// TwinCAT 3 PLC project AD_DA_V2
// ProgramVersion: 3.1.4020.2
// libraries:
//   Tc2_ControllerToolbox, * (Beckhoff Automation GmbH)
//   Tc2_Standard, * (Beckhoff Automation GmbH)
//   Tc2_System, * (Beckhoff Automation GmbH)
//   Tc3_Module, * (Beckhoff Automation GmbH)
//   VisuDialogs, * (System)
// project tree:
//   FB_Lib/Conversion/ FB_ConfigAnalog.TcPOU, FB_Ia.TcPOU, FB_Qa.TcPOU, ST_MinMax.TcDUT
//   FB_Lib/FB_ActionneurSimple/ FB_ActionneurSimple.TcPOU, ST_Erreur.TcDUT, ST_ParamActionneur.TcDUT
//   FB_Lib/ FB_analo_and_digital.TcPOU, FB_Etape.TcPOU
//   FB_Lib/FB_GestionModes/ FB_Btn.TcPOU, FB_CycleAuto.TcPOU, FB_CycleInit.TcPOU, FB_CycleMan.TcPOU, FB_MMA.TcPOU, p_InitVar.TcPOU
//   FB_Lib/FB_GestionModes/IO/ ST_IO.TcDUT, ST_IOInput.TcDUT, ST_IOInputSimul.TcDUT, ST_IOOutput.TcDUT, ST_IOOutputSimul.TcDUT
//   FB_Lib/FB_GestionModes/Param/ E_ModeMMA.TcDUT, ST_Param.TcDUT, ST_ParamFixed.TcDUT, ST_ParamRecipe.TcDUT, ST_ParamStatus.TcDUT
//   / GlobalTextList.TcGTLO, PlcTask.TcTTO, Visualisierungsmanager.TcVMO (not stored)
//   GVLs/ GVL.TcGVL
//   POUs/ MAIN.TcPOU
//   VISUs/ vi_ConvertAnalog.TcVIS, vi_ConvertAnalog_1.TcVIS
// (motion and I/O tree: see PLC project 1calcul)
// real-time tasks:
//   TASK PlcTask: cycle T#1ms, priority 20, ADS port 350
// variable links:
//   AD-DA_V2/AD-DA_V2 Instance <-> Device 2 (EtherCAT)/Box 1 (BK1150)
//     PlcTask Inputs/GVL.fbIa.IaEntree <-> Term 4 (KL3404)/Channel 2/Daten Ein
//     PlcTask Outputs/GVL.fbQa.QaSortie <-> Term 5 (KL4434)/Channel 2/Daten Aus

CONFIGURATION AD_DA_V2
    RESOURCE PLC ON TwinCAT3
        TASK PlcTask(INTERVAL := T#10ms, PRIORITY := 20);
        PROGRAM MAIN WITH PlcTask : MAIN;
    END_RESOURCE
END_CONFIGURATION

// ---- FB_Lib/Conversion/ST_MinMax.TcDUT
TYPE ST_MinMax :
STRUCT
	lrMin: LREAL;
	lrMax: LREAL;
END_STRUCT
END_TYPE

// ---- FB_Lib/FB_ActionneurSimple/ST_Erreur.TcDUT
TYPE ST_Erreur :
STRUCT
	xState:BOOL; 		//shows the current error state
	iId : INT; 			//error number currently active
	sMessage : STRING; 	//error message for the active error
END_STRUCT
END_TYPE

// ---- FB_Lib/FB_ActionneurSimple/ST_ParamActionneur.TcDUT
TYPE ST_ParamActionneur :
STRUCT
	tTimeOut : TIME; 			//max time allowed for moving to position bevor xState=TRUE
	xPresenceSensOut : BOOL; 	//If at the out-pos a Sensor is available
	xPresenceSensIn : BOOL; 	//If at the in-pos a Sensor is availaible
	tMoveOutTimeDelay : TIME; 	//delay after activating xPresenceSensOut before turning off output. When there is no Sensor, only this time will be used.
	tMoveInTimeDelay : TIME; 	//delay after activating xPresenceSensIn before turning off output. When there is no Sensor, only this time will be used.
END_STRUCT
END_TYPE

// ---- FB_Lib/FB_GestionModes/IO/ST_IO.TcDUT
TYPE ST_IO :
STRUCT
	stIn:ST_IOInput;
	stOut:ST_IOOutput;
END_STRUCT
END_TYPE

// ---- FB_Lib/FB_GestionModes/IO/ST_IOInput.TcDUT
TYPE ST_IOInput :
STRUCT
	IxAruIO AT%I*  :BOOL;
	xStartIO AT%I* :BOOL;
	xStopIO AT%I*  :BOOL;
	xResetIO AT%I* :BOOL;
	xAuto AT%I* : BOOL;
	xManual AT%I* : BOOL;
END_STRUCT
END_TYPE

// ---- FB_Lib/FB_GestionModes/IO/ST_IOInputSimul.TcDUT
TYPE ST_IOInputSimul :
STRUCT
	IxAru :BOOL;
END_STRUCT
END_TYPE

// ---- FB_Lib/FB_GestionModes/IO/ST_IOOutput.TcDUT
TYPE ST_IOOutput :
STRUCT
	QxLampeRouge AT%Q*:BOOL;
	QxLampeVerte AT%Q* : BOOL;
	QxLampeOrange AT%Q* :BOOL;
END_STRUCT
END_TYPE

// ---- FB_Lib/FB_GestionModes/IO/ST_IOOutputSimul.TcDUT
TYPE ST_IOOutputSimul :
STRUCT
	QxLampeRouge AT%Q*:BOOL;
END_STRUCT
END_TYPE

// ---- FB_Lib/FB_GestionModes/Param/E_ModeMMA.TcDUT

TYPE E_ModeMMA :
(
	Init := 0,
	Auto,
	Man
);
END_TYPE

// ---- FB_Lib/FB_GestionModes/Param/ST_Param.TcDUT
TYPE ST_Param :
STRUCT
	stStatus:ST_ParamStatus;//informations d'états (compteur de pièces, modes,...)
	stFixed:ST_ParamFixed;//Paramètres pas en lien avec le produit, fixe
	stRecipe:ST_ParamRecipe;//Paramètres en lien avec le produit
END_STRUCT
END_TYPE

// ---- FB_Lib/FB_GestionModes/Param/ST_ParamFixed.TcDUT
TYPE ST_ParamFixed :
STRUCT
END_STRUCT
END_TYPE

// ---- FB_Lib/FB_GestionModes/Param/ST_ParamRecipe.TcDUT
TYPE ST_ParamRecipe :
STRUCT
	
END_STRUCT
END_TYPE

// ---- FB_Lib/FB_GestionModes/Param/ST_ParamStatus.TcDUT
TYPE ST_ParamStatus :
STRUCT
	eMMA : E_ModeMMA; 
	xModePasAPas:BOOL;
	xErreur:BOOL;
	xInitOk:BOOL;//indique que l'initialisation a été exécutée
END_STRUCT
END_TYPE

// ---- GVLs/GVL.TcGVL

VAR_GLOBAL
		fbQa:FB_Qa;
		fbIa:FB_Ia;
END_VAR

// ---- POUs/MAIN.TcPOU
PROGRAM MAIN
VAR
	Consigne: LREAL;
	deltaConsigne :LREAL;
	PID : FB_CTRL_PID;
	
END_VAR

fbQa();
fbIa();




PID.fSetpointValue:=Consigne;
PID.fActualValue:=fbIa.lrValeur;
PID.eMode:=2;

PID(fOut=>fbQa.lrConsigne,stParams.fKp:=2,stParams.tTn:=T#10S,stParams.tTv:=T#10S,stParams.tTd:=T#10S,stParams.fOutMaxLimit:=10,stParams.fOutMinLimit:=-10,stParams.bARWOnIPartOnly:=FALSE,
stParams.bDInTheFeedbackPath:=TRUE,stParams.bPInTheFeedbackPath:=TRUE,stParams.tCtrlCycleTime:=T#10MS,stParams.tTaskCycleTime:=T#10MS);

END_PROGRAM

// ---- FB_Lib/Conversion/FB_Qa.TcPOU
FUNCTION_BLOCK FB_Qa
VAR_INPUT
	///consigne dans l'unité de l'utilisateur, selon min et max de fbCongig.stValeur
	lrConsigne: LREAL;
	///configuration de la sortie analogique
	fbConfig: FB_ConfigAnalog;
END_VAR
VAR_OUTPUT
	///sortie analogique, atention, supprimer MatchingSize lors de la liaison avec la borne
	QaSortie AT %Q*: DINT;
	///écart de précision sur la valeur de consigne => valeur +/- écart
	lrEcart: LREAL;
	///tension en volt
	lrTension: LREAL;
END_VAR

// 
QaSortie:=fbConfig.mConvertValToAn(lrConsigne,lrTension=>lrTension,lrEcart=>lrEcart);

END_FUNCTION_BLOCK

// ---- FB_Lib/Conversion/FB_ConfigAnalog.TcPOU
FUNCTION_BLOCK FB_ConfigAnalog
VAR_INPUT
	///nombre de bit de la variable de transit du bus de terrain
	uiNbreBitBus: UINT;
	///nombre de bit du convertiseur Analogique/digital 
	uiNbreBitConv: UINT;
	///valeur min et max de la tension
	stTension: ST_minMax;
	///valeur min et max de la consigne
	stValeur: ST_minMax;
END_VAR
VAR
	udiNbreIncBus: UDINT;
	lrTemp: LREAL;
	///nombre d'incrément avant décalage d'offset sur valeur de consigne
	lrValInc: LREAL;
END_VAR

METHOD mCalculDelta : LREAL
VAR_INPUT
	stMinMax: ST_MinMax;
END_VAR
mCalculDelta:=stMinMax.lrMax-stMinMax.lrMin;
END_METHOD

METHOD mCalculInc : UDINT
VAR_INPUT
	uiNbreBitBus: UDINT;
END_VAR

mCalculInc:=SHL(1,uiNbreBitBus);
//mCaclulInc:=EXPT(2,uiNbreBitBus);
END_METHOD

METHOD mConvertAnToVal : LREAL
VAR_INPUT
	///valeur de consigne
	lrAna: LREAL;
END_VAR
VAR_OUTPUT
	///tension de la borne de sortie
	lrTension: LREAL;
	///Ecart de l'escalier sur la borne de sortie en unité de valeur
	lrEcart: LREAL;
END_VAR
VAR
	lrValeur: LREAL;
END_VAR
//vérification que lrVal compris entre min et max
(*IF lrVal>stValeur.lrMax THEN
	lrVal:=stValeur.lrMax;
END_IF
IF lrVal>stValeur.lrMin THEN
	lrVal:=stValeur.lrMin;
END_IF*)
(*
lrVal:=MAX(lrVal,stValeur.lrMax);
lrVal:=MIN(lrVal,stValeur.lrMin);
*)


//Calcul du nombre d'incréments
udiNbreIncBus:=mCalculInc(uiNbreBitBus);
//Conversion de la valeur vers le résultat
//deltaTension/Nbreinc <-> deltaVal/Nbreinc val
lrValeur:=0;//réponse = 0 si hors condition
IF mCalculDelta(stValeur)<>0 THEN
	//décalage selon min max de la tension
	//IF stTension.lrMin<0 THEN
	//	//ajout de l'offset si min négatif
	//	lrTemp:=lrValInc-udiNbreIncBus/2-1;
	//	ELSE
	//	lrTemp:=lrValInc;
	//END_IF
	//nombre d'incréments par rapport à lrVal, avec décalage de stValeur.lrMin
	//lrValeur:=(lrAna*mCalculDelta(stValeur)-stValeur.lrMin)/udiNbreIncBus;
	//lrValInc:=udiNbreIncBus*(lrVal-stValeur.lrMin)/mCalculDelta(stValeur);
	//temp:=(iValMax-iValMin) / temp2;
	//oPhysicalValue:=iValMin + (temp * (iRAWValue+temp2/2));
	lrValeur:=(mCalculDelta(stValeur)/udiNbreIncBus)*lrAna;
	
END_IF
//résultat de la méthode
mConvertAnToVal:=lrValeur;
//calcul de l'incrément tension
lrEcart:=(mCalculDelta(stTension)/udiNbreIncBus);
//résultat en unitée de tension
lrTension:=lrValInc*lrEcart+stTension.lrMin;
END_METHOD

METHOD mConvertValToAn : DINT
VAR_INPUT
	///valeur de consigne
	lrVal: LREAL;
END_VAR
VAR_OUTPUT
	///tension de la borne de sortie
	lrTension: LREAL;
	///Ecart de l'escalier sur la borne de sortie en unité de valeur
	lrEcart: LREAL;
END_VAR
//vérification que lrVal compris entre min et max
(*IF lrVal>stValeur.lrMax THEN
	lrVal:=stValeur.lrMax;
END_IF
IF lrVal>stValeur.lrMin THEN
	lrVal:=stValeur.lrMin;
END_IF*)
(*
lrVal:=MAX(lrVal,stValeur.lrMax);
lrVal:=MIN(lrVal,stValeur.lrMin);
*)
lrVal:=LIMIT(stValeur.lrMin,lrVal,stValeur.lrMax);

//Calcul du nombre d'incréments
udiNbreIncBus:=mCalculInc(uiNbreBitBus);
//Conversion de la valeur vers le résultat
//deltaTension/Nbreinc <-> deltaVal/Nbreinc val
lrTemp:=0;//réponse = 0 si hors condition
IF mCalculDelta(stValeur)<>0 THEN
	//nombre d'incréments par rapport à lrVal, avec décalage de stValeur.lrMin
	lrValInc:=udiNbreIncBus*(lrVal-stValeur.lrMin)/mCalculDelta(stValeur);
	//décalage selon min max de la tension
	IF stTension.lrMin<0 THEN
		//ajout de l'offset si min négatif
		lrTemp:=lrValInc-udiNbreIncBus/2-1;
		ELSE
		lrTemp:=lrValInc;
	END_IF
END_IF
//résultat de la méthode
mConvertValToAn:=LREAL_TO_DINT(lrTemp);
//calcul de l'incrément tension
lrEcart:=(mCalculDelta(stTension)/udiNbreIncBus);
//résultat en unitée de tension
lrTension:=lrValInc*lrEcart+stTension.lrMin;
END_METHOD

END_FUNCTION_BLOCK

// ---- FB_Lib/Conversion/FB_Ia.TcPOU
FUNCTION_BLOCK FB_Ia
VAR_INPUT
	///configuration de la sortie analogique
	fbConfig: FB_ConfigAnalog;
END_VAR
VAR_OUTPUT
	///Valeur dans l'unité de l'utilisateur, selon min et max de fbCongig.stValeur
	lrValeur: LREAL;
	///sortie analogique, atention, supprimer MatchingSize lors de la liaison avec la borne
	IaEntree AT%I*: INT;
	///écart de précision sur la valeur de consigne => valeur +/- écart
	lrEcart: LREAL;
	///tension en volt
	lrTension: LREAL;
END_VAR
VAR
END_VAR

lrValeur:=fbConfig.mConvertAnToVal(IaEntree,lrTension=>lrTension,lrEcart=>lrEcart);

END_FUNCTION_BLOCK

// ---- FB_Lib/FB_ActionneurSimple/FB_ActionneurSimple.TcPOU
FUNCTION_BLOCK FB_ActionneurSimple
VAR_INPUT
	xInGoOut AT%I*:BOOL;				//input for going out
	xInGoIn AT%I*:BOOL;					//input for going in
	xReset AT%I*:BOOL;					//Reset all (go back to init state
	
	xAutorizeOut AT%I* : BOOL;		//allowed to do the move requested with xInGoOut, If this is false Programm will threw an error
	xAutorizeIn At%I* : BOOL;			//allowed to do the move requested with xInGoIn, If this is false Programm will threw an error
	
	stParam:ST_ParamActionneur;	//Param for actuator 
END_VAR
VAR_OUTPUT
	xInOutPos:BOOL;
	xInInPos:BOOL;
	
	xGoingOutNow AT%Q*:BOOL; //indication that actor is going in Out-Pos
	xGoingInNow AT%Q*:BOOL; //indication that actor is going in In-Pos
	
	QxOutOutput AT%Q*:BOOL;//Output to actuator for going Out
	QxInOutput AT%Q*:BOOL;//Output to actuator for going In
	
	IxSensOut AT%I*:BOOL;	//Sensor for the reached In-Pos
	IxSensIn AT%I*:BOOL;//Sensor for the reached Out-Pos
		
	stError:ST_Erreur;//Error Struct
	
	QxVanneDeBloquage AT%Q* : BOOL; //Vanne de blocace. Elle devient seulement 1 si l'autorisation entree/sortie est present
END_VAR
VAR
	fbEtape:FB_Etape;
	fbTimeOut:TON;
	fbRTrigOut:R_Trig;
	fbRTrigIn:R_Trig;
		
	

END_VAR

fbEtape.mActualisation(xModeStepForStep,xNextStep);

//check rising edges on 
fbRTrigOut(clk:=xInGoOut);
fbRTrigIn(clk:=xInGoIn);

//Go to the next step when there is an Out-Command
IF fbRTrigOut.Q AND NOT(fbEtape.iNo>=200 AND fbEtape.iNo<=299) THEN	//When rising-edge was detected
	IF xAutorizeOut THEN
		fbEtape.piVal:=200;
	ELSE
		stError.iId:=10;
		stError.sMessage:='Autorisation refusee pour action sortir verin';
	END_IF		
fbEtape.piVal:=200;	
END_IF

//Go to the next step when there is an In-Command
IF fbRTrigIn.Q AND NOT(fbEtape.iNo>=100 AND fbEtape.iNo<=199) THEN	//When rising-edge was detected and not already going In
	IF xAutorizeIn THEN
		fbEtape.piVal:=100;
	ELSE
		stError.iId:=11;
		stError.sMessage:='Autorisation refusee pour action rentrer verin';
	END_IF	
END_IF

//Reset
IF xReset THEN
	fbEtape.piVal:=0;
	stError.xState:=0;
	xInOutPos:=0;
	xInInPos:=0;
END_IF

//check pour vanne de blocage
QxVanneDeBloquage:= (xAutorizeOut OR xAutorizeIn);

//Reset de l'erreur
IF stError.xState THEN
	stError.iId:=0;
	stError.sMessage:='';
END_IF



CASE fbEtape.iNo OF
	0:fbEtape.psMess:='Wait for an In or Out command';
	//-----------------------------------------------
	100:fbEtape.psMess:='Action go In';
		IF xAutorizeIn THEN
			fbEtape.piVal:=110;
			fbEtape.tTimeQ:=stParam.tMoveInTimeDelay;
		END_IF
	110:fbEtape.psMess:='Going in, waiting for IxSensIn';
		IF (IxSensIn AND stParam.xPresenceSensIn) OR NOT stParam.xPresenceSensIn THEN
			fbEtape.piVal:=150;
		END_IF
	150:fbEtape.psMess:='Action rentre, attend tenps d enveloppe';
		IF fbEtape.xTimeQ THEN
			fbEtape.piSVal:=199;
		END_IF
	199:fbEtape.psMess:='In-Position reached';
		IF (NOT IxSensIn) AND stParam.xPresenceSensIn THEN
			fbEtape.piVal:=150;
		END_IF
	//-----------------------------------------------
	200:fbEtape.psMess:='Action go Out';
		IF xAutorizeOut THEN
			fbEtape.piVal:=210;
			fbEtape.tTimeQ:=stParam.tMoveInTimeDelay;
		END_IF
	210:fbEtape.psMess:='Going Out, waiting for IxSensOut';
		IF (IxSensOut AND stParam.xPresenceSensOut) OR NOT stParam.xPresenceSensOut THEN
			fbEtape.piVal:=250;
		END_IF
	250:fbEtape.psMess:='Action sort, attend temps d enveloppe';
		IF fbEtape.xTimeQ THEN
			fbEtape.piSVal:=299;
		END_IF
	299:fbEtape.psMess:='Out-Pos reached';
		IF (NOT IxSensOut) AND stParam.xPresenceSensoUT THEN
			fbEtape.piVal:=250;
		END_IF
	
	999:fbEtape.psMess:='Erreur';
END_CASE

//Activation du Timer
fbTimeOut(IN:=(fbEtape.iNo>100 AND fbEtape.iNo<199 OR fbEtape.iNo>200 AND fbEtape.iNo<299)
				AND (NOT fbRTrigIn.Q AND NOT fbRTrigOut.Q),PT:=stParam.tTimeOut);	


(*Liste des erreurs possibles :
-	10 Si un ordre de déplacement sort est donné et que l’entrée, xAutoriseSort n’est pas vrai, on indique une erreur
-	11 Idem pour xAutoriseRentre
-	20 Erreur de timeout sort
-	21 Erreur de timeout rentre
-	30 Les deux fins de course sont vraies en même temps
-	31 Double consignes, xSetSort=1 et xSetRentre=1*)				
//Gestion des erreurs
IF fbTimeOut.Q THEN
	IF fbEtape.iNo < 200 THEN
		stError.sMessage:='Erreur de timeout rentre';
		stError.iId:=21;
	ELSIF fbEtape.iNo>200 THEN
		stError.sMessage:='Erreur de timeout sort';
		stError.iId:=20;
	END_IF
ELSIF IxSensIn AND IxSensOut THEN
	stError.sMessage:='Les deus fins de course sont vraies en même temps';
	stError.iId:=30;
ELSIF xInGoOut AND xInGoIn THEN
	stError.sMessage:='Double consigne,xSetSort=1 et xSetRentre=1';
	stError.iId:=31;
END_IF

stError.xState :=fbEtape.iNo=999 OR fbTimeOut.Q OR (IxSensIn AND IxSensOut) OR (xInGoIn AND xInGoOut);


//Activation des états
xInInPos:=fbEtape.iNo=199;
xInOutPos:=fbEtape.iNo=299;
xGoingInNow:= QxInOutput AND NOT IxSensIn;
xGoingOutNow:= QxOutOutput AND NOT IxSensOut;


//Activation des sorties
QxOutOutput:=fbEtape.iNo>200 AND fbEtape.iNo<=299;
QxInOutput:=fbEtape.iNo>100 AND fbEtape.iNo<=199;

END_FUNCTION_BLOCK

// ---- FB_Lib/FB_Etape.TcPOU
FUNCTION_BLOCK FB_Etape
VAR_INPUT
	tTimeQ :TIME;			//Time to stay in one state after which xTimeQ will go to TRUE
END_VAR
VAR_OUTPUT
	tTimeState: TIME ; 	//passed time in the actual state
	xTimeQ : BOOL ;		//is TRUE when time passed in the actual State is greather then tTimeQ
	xTransition:BOOL; 	//information that the state has just changed. For use when entering a new State the first time
	iNo:INT:=0; 		//State number running at the moment
	sMess :STRING ; 	//Information message about the current running state
END_VAR
VAR
	iMemNo:INT;				//Used for xTransition. Saves the actual state of the machine
	fbTon:ton;				//Timer for the actual State
	fbRtrig:R_trig;			//detector for rising edges
	xMemModeStepByStep:BOOL;	//Mem for the actual running Mode (see method mActualisation)
	
END_VAR

//executed at each state-machine-loop
METHOD PUBLIC mActualisation
VAR_INPUT
	xModeStepByStep: BOOL; //activate the Stepping-Mode (TRUE=ON)
	xSetNextStep: BOOL; //go to the next Step on rising eddge
END_VAR
//manage StepByStep
//-----------------

//Detect rising edge
fbRtrig(CLK:=xSetNextStep);
//copy the mode input to use it in piSVal
xMemModeStepByStep:=xModeStepByStep;

//detect a state changement in the state machine
xTransition:=iNo<>iMemNo;

//start Method when the state has changed
IF xTransition THEN
	mTransition();
END_IF

//manage the Timer and associated Variabels
//-----------------------------------------
fbTON(IN:=(iNo=iMemNo), PT:=T#71582M47S295MS, ET=>tTimeState); //will be resetted when the state is changed

//going to TRUE when longer in the actual State than tTimeQ
xTimeQ:=(tTimeState>=tTimeQ);

//save the last running state
iMemNo:=iNo;
END_METHOD

//Executed when a State has changed
METHOD PRIVATE mTransition
//make a new String to display
sMess:=CONCAT('iNo:=',int_to_string(iNo));
END_METHOD

//going to the next step while paying attention to StepByStep Mode
PROPERTY PUBLIC piSVal : INT
SET
IF NOT xMemModeStepByStep THEN
	//Step by step mode is off
	iNo:=piSVal;
	ELSIF fbRtrig.Q THEN
		//a button press on "xSetNextStep" has been detected
		iNo:=piSVal;
END_IF
END_SET
END_PROPERTY

//going to the next step without paying attention to StepByStep Mode
PROPERTY PUBLIC piVal : INT
SET
//set the next step
iNo:=piVal;
END_SET
END_PROPERTY

//
PROPERTY PUBLIC psMess : STRING
SET
//write the description of the actual step to sMess
IF xTransition THEN
	sMess:=psMess;
END_IF
END_SET
END_PROPERTY

END_FUNCTION_BLOCK

// ---- FB_Lib/FB_analo_and_digital.TcPOU
FUNCTION_BLOCK FB_analo_and_digital
VAR_INPUT
	iRAWValue : LREAL;			//raw Value read from sensor (registre)
	iResolution : INT; 		//resolution in bits
	iValMin: INT;			//min physical value possible
	iValMax: INT;			//max physical value possible
	iTransToPhysical : BOOL;	//RAW --> Physical when TRUE
	iPhysical2Value: LREAL; 	//valeur physique (ex tr/min)
	iValInputMax: INT;		//max input value at the Box
	iValInputMin: INT;		//min input value at the Box
	iPhysicalValue : LREAL;	//valeur physique sur l'entree de l'input
END_VAR
VAR_OUTPUT
	oValInputMin: INT;		//min input value at the Box
	oPhysicalValue : LREAL;	//valeur physique sur l'entree de l'input
	oInputValue : LREAL;	//valeur physique sur l'entree de l'input
	oPhysical2Value: LREAL; 	//valeur physique (ex tr/min)
	oRAWValue : LREAL;			//raw Value read from sensor (registre)
END_VAR
VAR	
	temp : LREAL;
	temp2 : LREAL;	
END_VAR

temp2:=expt(2,iResolution);



IF(iTransToPhysical) THEN
	//RAW Input to physical value
	temp:=(iValInputMax-iValInputMin) / temp2;
	oInputValue:=iValInputMin + (temp * (iRAWValue + temp2/2));
	
	
	temp:=(iValMax-iValMin) / temp2;
	oPhysicalValue:=iValMin + (temp * (iRAWValue+temp2/2));
ELSE
	//Physical value to raw-Value
	temp:=(iValMax-iValMin) / temp2;
	oRAWValue:= iValMin+ (iPhysicalValue / temp);
			
END_IF

END_FUNCTION_BLOCK

// ---- FB_Lib/FB_GestionModes/FB_Btn.TcPOU
FUNCTION_BLOCK FB_Btn
VAR_INPUT
	xStart:BOOL;
	xStop:BOOL;
	xReset:BOOL;
	xNextPas:BOOL;
	xAru:BOOL;
	
	xManAct1Rentre: BOOL;
	xManAct1Sort : BOOL;
	
	xManAct2Rentre: BOOL;
	xManAct2Sort : BOOL;
	
	xManAct3Rentre: BOOL;
	xManAct3Sort : BOOL;
END_VAR
VAR_OUTPUT
END_VAR
VAR
END_VAR

END_FUNCTION_BLOCK

// ---- FB_Lib/FB_GestionModes/FB_CycleAuto.TcPOU
FUNCTION_BLOCK FB_CycleAuto
VAR_INPUT
	xStart:BOOL;
	xStop:BOOL;
	xReset:BOOL;
END_VAR
VAR_OUTPUT
	fbRtrigStart:R_trig;
	xBusy:BOOL;
	xMemStop:BOOL:=FALSE;
	iEtape:INT;
END_VAR
VAR
	fbEtape:FB_Etape;
END_VAR

fbEtape.mActualisation(stParam.stStatus.xModePasAPas,fbBtn.xNextPas);

fbRtrigStart(clk:=xStart);

IF xStop THEN
	xMemStop:=TRUE;
END_IF

IF xReset THEN
	fbEtape.piVal:=0;
END_IF

CASE fbEtape.iNo OF
	0:IF fbRtrigStart.Q THEN
		xMemStop:=FALSE;
		fbEtape.piVal:=100;
	END_IF
	100:fbEtape.psMess:='fonction allume lampe1';
		//assigne le temps de comptage
		fbEtape.tTimeQ:=T#2S;
		fbEtape.piVal:=110;
	110:fbEtape.psMess:='activation compteur 2s - attendre fin comptage';
		IF fbEtape.xTimeQ THEN
			fbEtape.piSVal:=120;
		END_IF
	120:fbEtape.psMess:='Actionneur1 sort';
		IF fbAct1.xInOutPos THEN
			fbEtape.piSVal:=121;
		END_IF
	121:fbEtape.psMess:='Actionneur2 sort';
		IF fbAct2.xInOutPos THEN
			fbEtape.piSVal:=122;
		END_IF
	122:fbEtape.psMess:='Actionneur3 sort';
		IF fbAct3.xInOutPos THEN
			fbEtape.piSVal:=130;
		END_IF
	130:fbEtape.psMess:='Actionneur3 rentre';
		IF fbAct3.xInInPos THEN
			fbEtape.piSVal:=131;
		END_IF
	131:fbEtape.psMess:='Actionneur2 rentre';
		IF fbAct2.xInInPos THEN
			fbEtape.piSVal:=132;
		END_IF
	132:fbEtape.psMess:='Actionneur1 rentre';
		IF fbAct1.xInInPos THEN
			fbEtape.piSVal:=200;
		END_IF
	200:fbEtape.psMess:='fonction allume lampe1';
		//assigne le temps de comptage
		fbEtape.tTimeQ:=T#1S;
		fbEtape.piVal:=210;
	210:fbEtape.psMess:='activation compteur 1s - attendre fin comptage';
		IF fbEtape.xTimeQ THEN
			fbEtape.piSVal:=300;
		END_IF
	300:fbEtape.psMess:='fonction lampes off';
		//assigne le temps de comptage
		fbEtape.tTimeQ:=T#2S;
		fbEtape.piVal:=310;
	310:fbEtape.psMess:='activation compteur 2s - attendre fin comptage';
		IF fbEtape.xTimeQ THEN
			fbEtape.piSVal:=900;
		END_IF
	900:fbEtape.psMess:='Test si demande arrrêt en fin de cycle';
		IF xMemStop THEN
		fbEtape.piSVal:=999;
		ELSE
		fbEtape.piSVal:=100;
	END_IF
	999:fbEtape.psMess:='FIN';
		fbEtape.piSVal:=0;
END_CASE

xBusy:=fbEtape.iNo<>0;
iEtape:=fbEtape.iNo;

END_FUNCTION_BLOCK

// ---- FB_Lib/FB_GestionModes/FB_CycleInit.TcPOU
FUNCTION_BLOCK FB_CycleInit
VAR_INPUT
	xStart : BOOL;
	xStop : BOOL;
END_VAR
VAR_OUTPUT
	fbRtrigStart:R_trig;
	xBusy:BOOL;
	iEtape:INT;
END_VAR
VAR
	fbEtape:FB_Etape;
END_VAR

fbEtape.mActualisation(stParam.stStatus.xModePasAPas,fbBtn.xNextPas);

fbRtrigStart(clk:=fbBtn.xStart);


CASE fbEtape.iNo OF
	0:fbEtape.psMess:='Attendre - Pret';
		IF xStart THEN
			fbEtape.piVal:=99;
		END_IF
	99: fbEtape.psMess:='Reset sur les Actionneurs';
		fbEtape.piSVal:=100;
		
	100:fbEtape.psMess:='Initialiser les positions';
		IF  fbAct1.xInInPos AND fbAct2.xInInPos AND NOT fbAct3.xInInPos THEN
			fbEtape.piSVal:=999;
		END_IF
	
	999:fbEtape.psMess:='Fin Cycle Init - Attente de Stop';
		IF (xStop) THEN
		fbEtape.piSVal:=0;
	END_IF
END_CASE

xBusy:=fbEtape.iNo<>0;
iEtape:=fbEtape.iNo;

END_FUNCTION_BLOCK

// ---- FB_Lib/FB_GestionModes/FB_CycleMan.TcPOU
FUNCTION_BLOCK FB_CycleMan
VAR_INPUT
	xStart : BOOL;
	xStop : BOOL;
	
	
END_VAR
VAR_OUTPUT
	fbRtrigStart:R_trig;
	xBusy:BOOL;
	iEtape:INT;
END_VAR
VAR
	fbEtape:FB_Etape;
END_VAR

fbEtape.mActualisation(stParam.stStatus.xModePasAPas,fbBtn.xNextPas);

fbRtrigStart(clk:=fbBtn.xStart);


CASE fbEtape.iNo OF
	0:	fbEtape.psMess:='Attendre - Pret';
		IF xStart THEN
			fbEtape.piVal:=100;
		END_IF
	100:fbEtape.psMess:='Selectioner quoi faire';
		//changer de mode
		IF  stParam.stStatus.eMMA<>Man THEN
			fbEtape.piSVal:=990;
		END_IF
		//Act1:
		IF (fbBtn.xManAct1Rentre) THEN
			fbEtape.piVal:=201;
		END_IF
		IF (fbBtn.xManAct1Sort) THEN
			fbEtape.piVal:=202;
		END_IF
		//Act2:
		IF (fbBtn.xManAct2Rentre) THEN
			fbEtape.piVal:=203;
		END_IF
		IF (fbBtn.xManAct2Sort) THEN
			fbEtape.piVal:=204;
		END_IF
		//Act3:
		IF (fbBtn.xManAct3Rentre) THEN
			fbEtape.piVal:=205;
		END_IF
		IF (fbBtn.xManAct3Sort) THEN
			fbEtape.piVal:=206;
		END_IF
		
		
		
	201: fbEtape.psMess:='Action : Act 1 Rentre';
		IF (NOT fbBtn.xManAct1Rentre) THEN
			fbEtape.piVal:=100;
		END_IF
	202: fbEtape.psMess:='Action : Act 1 Sort';
		IF (NOT fbBtn.xManAct1Sort) THEN
			fbEtape.piVal:=100;
		END_IF
	203: fbEtape.psMess:='Action : Act 2 Rentre';
		IF (NOT fbBtn.xManAct2Rentre) THEN
			fbEtape.piVal:=100;
		END_IF
	204: fbEtape.psMess:='Action : Act 2 Sort';
		IF (NOT fbBtn.xManAct2Sort) THEN
			fbEtape.piVal:=100;
		END_IF
	205: fbEtape.psMess:='Action : Act 3 Rentre';
		IF (NOT fbBtn.xManAct3Rentre) THEN
			fbEtape.piVal:=100;
		END_IF
	206: fbEtape.psMess:='Action : Act 3 Sort';
		IF (NOT fbBtn.xManAct3Sort) THEN
			fbEtape.piVal:=100;
		END_IF
	
	990:fbEtape.psMess:='Finir Cycle Man';
		//ici on fait des choses de fin (ex. eteindre un moteur qui tourne encore)
		IF (1) THEN
			fbEtape.piSVal:=999;
		END_IF	
	999:fbEtape.psMess:='Fin Cycle Manuel';
		IF (xStop) THEN
			fbEtape.piSVal:=0;
		END_IF
		
END_CASE

xBusy:=fbEtape.iNo<>0;
iEtape:=fbEtape.iNo;

END_FUNCTION_BLOCK

// ---- FB_Lib/FB_GestionModes/FB_MMA.TcPOU
FUNCTION_BLOCK FB_MMA
VAR_INPUT
END_VAR
VAR_OUTPUT
	iEtape:INT;
END_VAR
VAR
	fbEtape:FB_Etape;
	p_InitVar : p_InitVar;
END_VAR

fbEtape.mActualisation(FALSE,FALSE);

//on active l'arret d'urgence si l'entree devient false
IF NOT fbBtn.xAru AND fbEtape.iNo>10 AND fbEtape.iNo<800 THEN
	fbEtape.piVal:=900; 
END_IF

//on fait un reset
IF fbBtn.xReset AND fbEtape.iNo>10 AND fbEtape.iNo<800 THEN
	fbEtape.piVal:=800;
END_IF


CASE fbEtape.iNo OF
	0://mise en marche du système
		fbEtape.piVal:=10;
	
	10://OB100 Siemens
		p_InitVar(); //initialiser les vars (propre a la machine)
		fbEtape.piVal:=50;
	
	50:fbEtape.psMess:='Selection du mode MMA';
		IF (stParam.stStatus.eMMA=Auto) THEN
			fbEtape.piVal:=300;
		ELSIF (stParam.stStatus.eMMA=Man) THEN
			fbEtape.piVal:=210;
		ELSIF (stParam.stStatus.eMMA=Init) THEN
			fbEtape.piVal:=100;
		END_IF
		
	//--------------------------------------------------------------
	//Init
	//--------------------------------------------------------------
	100:fbEtape.psMess:='Cycle Init | Attente de fbBtn.xStart';
		IF (fbBtn.xStart) THEN
			fbEtape.piVal:=110;
		ELSIF (stParam.stStatus.eMMA<>Init) THEN
			fbEtape.piVal:=50;
		END_IF
	110:fbEtape.psMess:='Cycle Init | Attente fin';
		IF fbCycleInit.iEtape=999 THEN
		fbEtape.piVal:=50;
		END_IF
	111:fbEtape.psMess:='Cycle Init | Finir';
		IF fbCycleInit.xBusy THEN
		fbEtape.piVal:=50;
		END_IF
		
	//--------------------------------------------------------------
	//Manual
	//--------------------------------------------------------------
	210:fbEtape.psMess:='Cycle Manuel | Attente de changement de mode';
		IF (fbCycleMan.iEtape=999) THEN
		fbEtape.piVal:=211;
		END_IF
	211:fbEtape.psMess:='Cycle Manuel | Finir';
		IF (fbCycleMan.xBusy) THEN
		fbEtape.piVal:=50;
		END_IF
		
	//--------------------------------------------------------------
	//Auto
	//--------------------------------------------------------------
	300:fbEtape.psMess:='Mode Auto | Attente de fbBtn.xStart';
		IF (fbBtn.xStart) THEN
			fbEtape.piVal:=340;
		ELSIF (stParam.stStatus.eMMA<>Auto) THEN
			fbEtape.piVal:=50;
		END_IF
	
	340:fbEtape.psMess:='Mode Auto | Cycle Init - attente fin';
		//si le cycle INIT est terminé alors on continue
		fbEtape.piVal:=341;
		
	341:fbEtape.psMess:='Mode Auto | Cycle Init - Finir';
		//si le cycle INIT est terminé alors on continue
		IF fbCycleInit.iEtape=999 THEN
			fbEtape.piVal:=350;
		END_IF
		
	350:fbEtape.psMess:='Mode Auto | Production - attend signal Stop';
		IF (fbBtn.xStop OR stParam.stStatus.xErreur ) THEN 
			fbEtape.piVal:=390;
		END_IF
		
	390:fbEtape.psMess:='Mode Auto | Attendre fin';
		IF (NOT fbCycleAuto.xBusy) THEN
			fbEtape.piVal:=50;
		END_IF
		
	//--------------------------------------------------------------
	//Reset
	//--------------------------------------------------------------
	800:fbEtape.psMess:='Reset | Procédure de reset, stop imédiat';
		fbEtape.piVal:=810;
	810:fbEtape.psMess:='Reset | Ordre pour pilotage reste sur cycle';
		fbEtape.piVal:=899;
	899:fbEtape.psMess:='Reset | Fin de procédure Reset';
		fbEtape.piVal:=50;
		
	//--------------------------------------------------------------
	//ARU
	//--------------------------------------------------------------
	900:fbEtape.psMess:='ARU | Procédure de ARU';
		fbEtape.piVal:=910;
	910:fbEtape.psMess:='ARU | Ordre pour pilotage reste sur cycle';
		fbEtape.piVal:=950;
	950:fbEtape.psMess:='ARU | ok - Attente de quittance';
		IF fbBtn.xAru THEN
			fbEtape.piVal:=999;
	END_IF
	999:fbEtape.psMess:='ARU | Fin de procédure ARU';
		fbEtape.piVal:=50;
END_CASE


iEtape:=fbEtape.iNo;

END_FUNCTION_BLOCK

// ---- FB_Lib/FB_GestionModes/p_InitVar.TcPOU
FUNCTION_BLOCK p_InitVar
VAR_INPUT
END_VAR
VAR_OUTPUT
END_VAR
VAR
	tEnvStabSort: INT;
END_VAR

fbAct1.stParam.xPresenceSensIn:=TRUE;
fbAct1.stParam.xPresenceSensOut:=TRUE;
fbAct1.stParam.tTimeOut:=T#10S;
fbAct1.stParam.tMoveInTimeDelay:=T#1.5S;
fbAct1.stParam.tMoveOutTimeDelay:=T#1.5S;

fbAct2.stParam.xPresenceSensIn:=TRUE;
fbAct2.stParam.xPresenceSensOut:=TRUE;
fbAct2.stParam.tTimeOut:=T#10S;
fbAct2.stParam.tMoveInTimeDelay:=T#1.5S;
fbAct2.stParam.tMoveOutTimeDelay:=T#1.5S;

fbAct3.stParam.xPresenceSensIn:=FALSE;
fbAct3.stParam.xPresenceSensOut:=TRUE;
fbAct3.stParam.tTimeOut:=T#10S;
fbAct3.stParam.tMoveInTimeDelay:=T#3S;
fbAct3.stParam.tMoveOutTimeDelay:=T#1.5S;

stParam.stStatus.eMMA:=Init;

END_FUNCTION_BLOCK

// ---- GlobalTextList.TcGTLO
TEXTLIST GlobalTextList
  0 = 'Consigne: %.2f'
  8 = 'fbConfig.lrTemp : %.2f'
  11 = 'fbConfig.lrValInc : %.2f'
  7 = 'fbConfig.udiNbreIncBus : %i'
  9 = 'lrEcart : %.5f'
  10 = 'lrTension : %.2f'
  15 = 'QaSortie : %2.5f'
  13 = 'QaSortie : %d'
  14 = 'QaSortie : %f'
  6 = 'QaSortie : %i'
  12 = 'QaSortie : %r'
  1 = 'stConfigBus.uiNbBits: %i'
  2 = 'stTension.lrMax : %.2f'
  3 = 'stTension.lrMin : %.2f'
  4 = 'stValeur.lrMax : %.2f'
  5 = 'stValeur.lrMin : %.2f'
END_TEXTLIST

// ---- VISUs/vi_ConvertAnalog.TcVIS
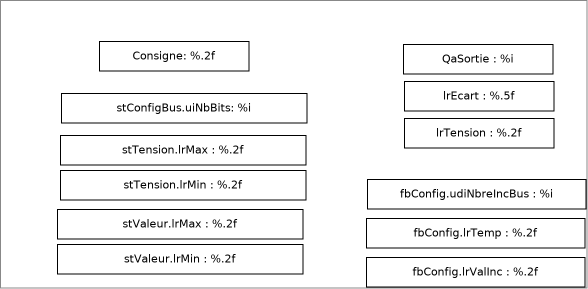
VISUALIZATION vi_ConvertAnalog  // 588x289
    Rectangle (99,41 150x30), "Consigne: %.2f", text variable: fbQa.lrConsigne
        OnMouseDown: write the text variable via Default
    Rectangle (61,93 246x30), "stConfigBus.uiNbBits: %i", text variable: fbQa.fbConfig.uiNbreBitBus
        OnMouseDown: write the text variable via Default
    Rectangle (60,135 246x30), "stTension.lrMax : %.2f", text variable: fbQa.fbConfig.stTension.lrMax
        OnMouseDown: write the text variable via Default
    Rectangle (60,170 246x30), "stTension.lrMin : %.2f", text variable: fbQa.fbConfig.stTension.lrMin
        OnMouseDown: write the text variable via Default
    Rectangle (57,209 246x30), "stValeur.lrMax : %.2f", text variable: fbQa.fbConfig.stValeur.lrMax
        OnMouseDown: write the text variable via Default
    Rectangle (57,244 246x30), "stValeur.lrMin : %.2f", text variable: fbQa.fbConfig.stValeur.lrMin
        OnMouseDown: write the text variable via Default
    Rectangle (403,44 150x30), "QaSortie : %i", text variable: fbQa.QaSortie
    Rectangle (367,179 219x30), "fbConfig.udiNbreIncBus : %i", text variable: fbQa.fbConfig.udiNbreIncBus
    Rectangle (366,218 219x30), "fbConfig.lrTemp : %.2f", text variable: fbQa.fbConfig.lrTemp
    Rectangle (404,81 150x30), "lrEcart : %.5f", text variable: fbQa.lrEcart
    Rectangle (404,118 150x30), "lrTension : %.2f", text variable: fbQa.lrTension
    Rectangle (366,257 219x30), "fbConfig.lrValInc : %.2f", text variable: fbQa.fbConfig.lrValInc
END_VISUALIZATION

// ---- VISUs/vi_ConvertAnalog_1.TcVIS
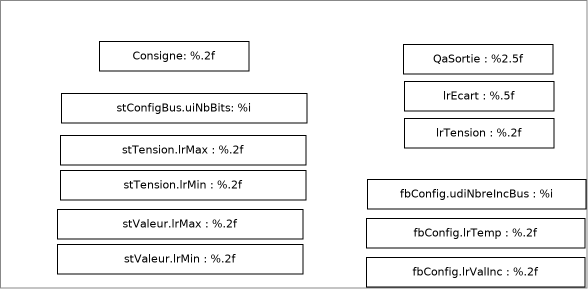
VISUALIZATION vi_ConvertAnalog_1  // 588x289
    Rectangle (99,41 150x30), "Consigne: %.2f", text variable: fbIa.IaEntree
        OnMouseDown: write the text variable via Default
    Rectangle (61,93 246x30), "stConfigBus.uiNbBits: %i", text variable: fbIa.fbConfig.uiNbreBitBus
        OnMouseDown: write the text variable via Default
    Rectangle (60,135 246x30), "stTension.lrMax : %.2f", text variable: fbIa.fbConfig.stTension.lrMax
        OnMouseDown: write the text variable via Default
    Rectangle (60,170 246x30), "stTension.lrMin : %.2f", text variable: fbIa.fbConfig.stTension.lrMin
        OnMouseDown: write the text variable via Default
    Rectangle (57,209 246x30), "stValeur.lrMax : %.2f", text variable: fbIa.fbConfig.stValeur.lrMax
        OnMouseDown: write the text variable via Default
    Rectangle (57,244 246x30), "stValeur.lrMin : %.2f", text variable: fbIa.fbConfig.stValeur.lrMin
        OnMouseDown: write the text variable via Default
    Rectangle (403,44 150x30), "QaSortie : %2.5f", text variable: fbIa.lrValeur
    Rectangle (367,179 219x30), "fbConfig.udiNbreIncBus : %i", text variable: fbIa.fbConfig.udiNbreIncBus
    Rectangle (366,218 219x30), "fbConfig.lrTemp : %.2f", text variable: fbIa.fbConfig.lrTemp
    Rectangle (404,81 150x30), "lrEcart : %.5f", text variable: fbIa.lrEcart
    Rectangle (404,118 150x30), "lrTension : %.2f", text variable: fbIa.lrTension
    Rectangle (366,257 219x30), "fbConfig.lrValInc : %.2f", text variable: fbIa.fbConfig.lrValInc
END_VISUALIZATION
